(* Logix 5000 project; controller cal1615 1756-L62 rev 20.11; software revision 20.05; part 20 of 81 *)
(* tags used below, declared in another part *)
   AFI : BOOL;   // Always False Bit
   FAULT : BOOL;   // Fault AFI
   p01_param_open_oven_temp : REAL;
   p01_param_oven_timer_presets : DINT[32];   // System Parameter Oven Timer Presets
   p01_recipe_active : recipe;   // Active Recipe
   p01_sys_enc : SYS_ENC;   // System Encoder
   p01r09_open_oven : BOOL;
   p01r09_pb_global_reset : BOOL;   // System Modes PB: Global Fault Reset
   p01r13_permissive_oxidizer : BOOL;   // System Line Start Sequence Permissive Oxidizer
   p02_dint_from_hmi : hmi_dint;
   p11_ai_tc01 : REAL;   // Zone 1 Analog Input Control Thermocouple 1
   p11_ai_tc02 : REAL;   // Zone 1 Analog Input Control Thermocouple 2
   p11_di_burner_auto : BOOL;   // Zone 1 Digital Input Burner Auto
   p11_di_burner_safeties_ok : BOOL;   // Zone 1 Digital Input Burner Safeties Ok
   p11_di_exh_flow_ok : BOOL;   // Zone 1 Digital Input Exhaust Flow OK
   p11_di_flame_on : BOOL;   // Zone 1 Digital Input Burner is On
   p11_di_recirc_flow_ok : BOOL;   // Zone 1 Digital Input Recirc Flow OK
   p11_param_fast_to_soak : REAL;   // Zone 1 Parameter Fast to Soak Control
   p11_param_pid1_ff : REAL;   // Zone 1 Parameter Fast PID Bias
   p11_param_pid1_kd : REAL;   // Zone 1 Parameter Fast PID Derivative Gain
   p11_param_pid1_ki : REAL;   // Zone 1 Parameter Fast PID Integral Gain
   p11_param_pid1_kp : REAL;   // Zone 1 Parameter Fast PID Proportional Gain
   p11_param_soak_to_fast : REAL;   // Zone 1 Parameter Soak to Fast Control
   p11r01 : routine;   // Zone 1 Main
   p11r02_shutdown_temp : BOOL;   // Zone 1 Misc Control Safe Shutdown Temperature
   p11r02_timer_safe_temp : TIMER[2];   // Zone 1 Misc Control Chamber SafeTemperature Dwell
   p11r10 : routine;   // Zone 1
   p11r10_timer_fault : TIMER[4];   // Zone 1 Fault Delay
   p11r10_timer_warning : TIMER[4];   // Zone 1 Warning Delay
   p11r12_Oven_auto_run_on : BOOL;   // Zone 1 Temp Sequence Oven Auto Run On
   p11r20 : routine;   // Zone 1 Temp Sequence
   p11r20_safeties_ok : BOOL;   // Zone 1 Temperature Control Burner Safeties OK this Lightoff
   p11r20_state : DINT;   // Zone 1 Temperature Control State
   p11r20_status : DINT;   // Zone 1 Temperature Control Sequence Status
   p11r20_timer_fault : TIMER[4];   // Zone 1 Temp Sequence Fault Delay
   p11r20_timer_state_11 : TIMER;   // Zone 1 Temp Sequence State 11 Dwell
   p11r20_timer_state_3 : TIMER;   // Zone 1 Temperature Control State 3 Dwell
   p11r20_timer_state_4 : TIMER;   // Zone 1 Temp Sequence State 4 Dwell
   p11r20_timer_state_7 : TIMER;   // Zone 1 Temp Sequence State 7 Dwell
   p11r20_timer_warning : TIMER[4];   // Zone 1 Temp Sequence Warning Delay
   p11r30 : routine;   // Zone 1 Temperature Control
   p11r30_cv_man_sp : REAL;   // Zone 1 Temperature Control Manual Heat Control Valve Setpoint
   p11r30_pb_auto : BOOL;   // Zone 1 Temperature Control PB: Zone Control Auto
   p11r30_pb_manual : BOOL;   // Zone 1 Temperature Control PB: Zone Control Manual
   p11r30_pb_zone_off : BOOL;   // Zone 1 Temperature Control PB: Stop Zone Heat Control
   p11r30_pb_zone_on : BOOL;   // Zone 1 Temperature Control PB: Start Zone Heat Control
   p11r30_permissive_run : BOOL;   // Zone 1 Temperature Control Run Permissive
   p11r30_pid_temp : PID;   // Zone 1 Temperature Control PID
   p11r30_pid_temp_pv : REAL;   // Zone 1 Temperature Control PID Temp Process Variable
   p11r30_pid_temp_sp : REAL;   // Zone 1 Temperature Control PID Temperature Control Setpoint
   p11r30_pid_temp_sp_error : REAL;   // Zone 1 Temperature Control Setpoint/Process Variable Error (ABS)
   p11r30_pid_temp_sp_last : REAL;   // Zone 1 Temperature Control Setpoint Last Scan
   p11r30_request_deviation_warning : BOOL;   // Zone 1 Temperature Control Request Setpoint Deviation Warning
   p11r30_request_heat : BOOL;   // Zone 1 Temperature Control Request Heat
   p11r30_request_heat_last : BOOL;   // Zone 1 Temperature Control Request Heat Last Scan
   p11r30_request_manual : BOOL;   // Zone 1 Temperature Control Request Manual Control
   p11r30_request_PID_shot : BOOL;
   p11r30_request_soak_control : BOOL;   // Zone 1 Temperature Control Request Soak Control
   p11r30_temp_deviation_setpoint : DINT;
   p11r30_timer_warning : TIMER[12];   // Zone 1 Temperature Control Warning Delay
   p11r30_vfds_ok : BOOL;
   p11r31 : routine;   // Zone 1 Exhaust VFD
   p11r32 : routine;   // Zone 1 Recirc VFD
   p12r30 : routine;   // Zone 2 Temperature Control
   p23_di_impreg_exhaust_running : BOOL;
   p23_di_impreg_tank_up : BOOL;   // Input Impreg Dip Tank Up
   p23r02 : routine;   // Impreg Misc Control
   p23r13 : routine;
(* P11_Zone_1, continued *)

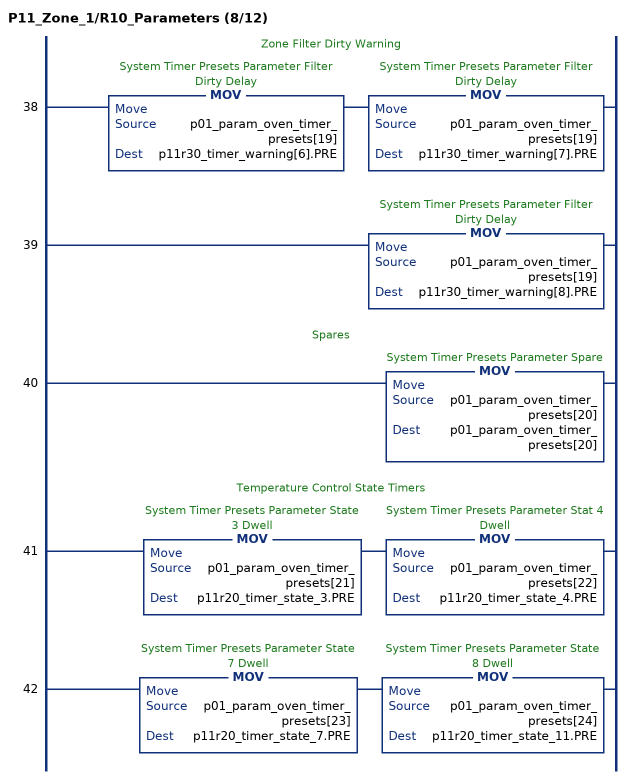
   [picture p305: P11_Zone_1/R10_Parameters rungs 38-42]
   // Zone Filter Dirty Warning
   38: MOV(p01_param_oven_timer_presets[19],p11r30_timer_warning[6].PRE)MOV(p01_param_oven_timer_presets[19],p11r30_timer_warning[7].PRE);
   39: MOV(p01_param_oven_timer_presets[19],p11r30_timer_warning[8].PRE);
   // Spares
   40: MOV(p01_param_oven_timer_presets[20],p01_param_oven_timer_presets[20]);
   // Temperature Control State Timers
   41: MOV(p01_param_oven_timer_presets[21],p11r20_timer_state_3.PRE)MOV(p01_param_oven_timer_presets[22],p11r20_timer_state_4.PRE);
   42: MOV(p01_param_oven_timer_presets[23],p11r20_timer_state_7.PRE)MOV(p01_param_oven_timer_presets[24],p11r20_timer_state_11.PRE);
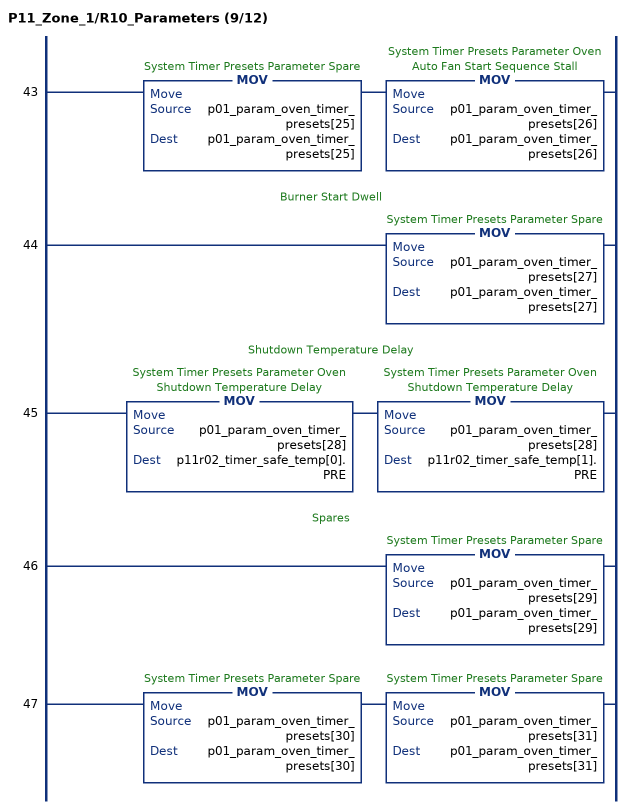
   43: MOV(p01_param_oven_timer_presets[25],p01_param_oven_timer_presets[25])MOV(p01_param_oven_timer_presets[26],p01_param_oven_timer_presets[26]);
   // Burner Start Dwell
   44: MOV(p01_param_oven_timer_presets[27],p01_param_oven_timer_presets[27]);
   // Shutdown Temperature Delay
   45: MOV(p01_param_oven_timer_presets[28],p11r02_timer_safe_temp[0].PRE)MOV(p01_param_oven_timer_presets[28],p11r02_timer_safe_temp[1].PRE);
   // Spares
   46: MOV(p01_param_oven_timer_presets[29],p01_param_oven_timer_presets[29]);
   47: MOV(p01_param_oven_timer_presets[30],p01_param_oven_timer_presets[30])MOV(p01_param_oven_timer_presets[31],p01_param_oven_timer_presets[31]);
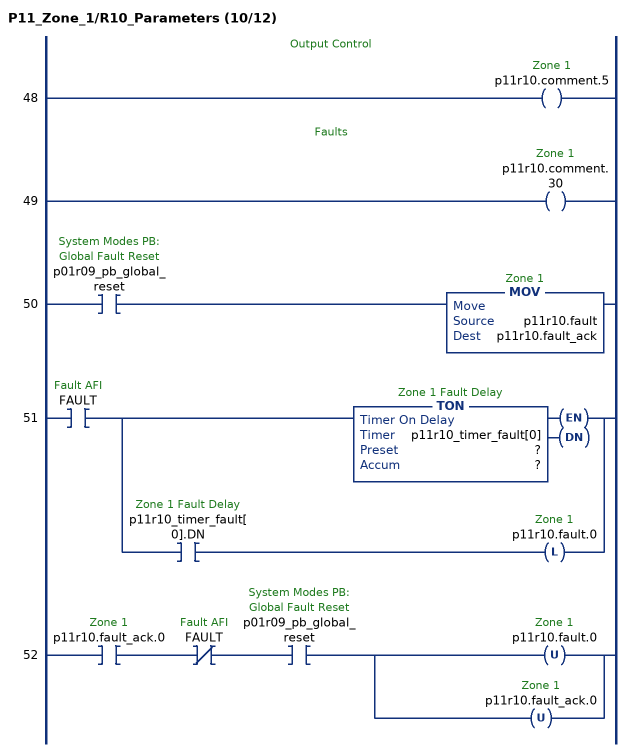
   // Output Control
   48: OTE(p11r10.comment.5);
   // Faults
   49: OTE(p11r10.comment.30);
   50: XIC(p01r09_pb_global_reset)MOV(p11r10.fault,p11r10.fault_ack);
   51: XIC(FAULT)[TON(p11r10_timer_fault[0],?,?) ,XIC(p11r10_timer_fault[0].DN) OTL(p11r10.fault.0) ];
   52: XIC(p11r10.fault_ack.0)XIO(FAULT)XIC(p01r09_pb_global_reset)[OTU(p11r10.fault.0) ,OTU(p11r10.fault_ack.0) ];
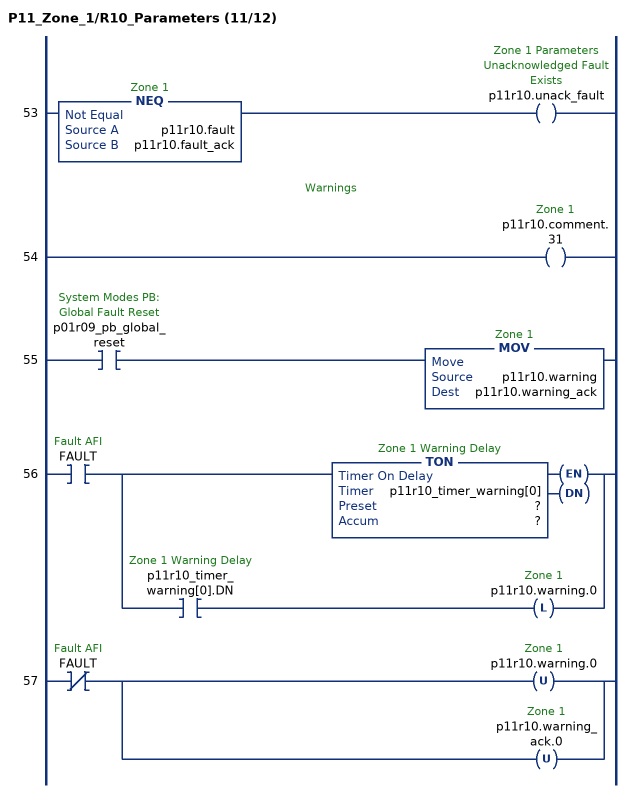
   53: NEQ(p11r10.fault,p11r10.fault_ack)OTE(p11r10.unack_fault);
   // Warnings
   54: OTE(p11r10.comment.31);
   55: XIC(p01r09_pb_global_reset)MOV(p11r10.warning,p11r10.warning_ack);
   56: XIC(FAULT)[TON(p11r10_timer_warning[0],?,?) ,XIC(p11r10_timer_warning[0].DN) OTL(p11r10.warning.0) ];
   57: XIO(FAULT)[OTU(p11r10.warning.0) ,OTU(p11r10.warning_ack.0) ];
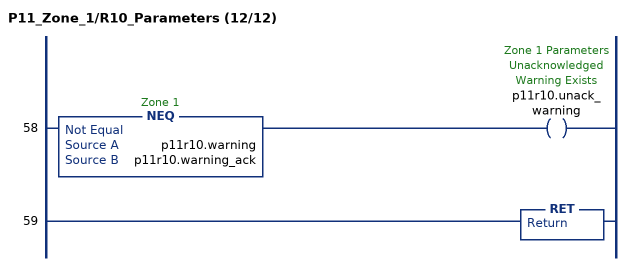
   58: NEQ(p11r10.warning,p11r10.warning_ack)OTE(p11r10.unack_warning);
   59: RET();
END_ROUTINE

ROUTINE R20_Temp_Sequence   (* ladder *)
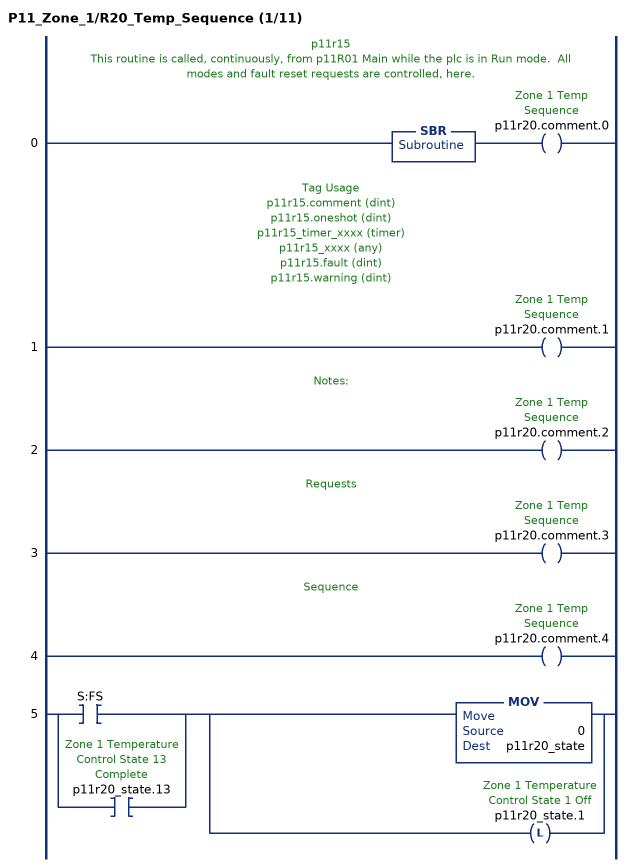
   // p11r15
   // This routine is called, continuously, from p11R01 Main while the plc is in Run mode.  All modes and fault reset requests are controlled, here.
   0: SBR()OTE(p11r20.comment.0);
   // Tag Usage
   // p11r15.comment (dint)
   // p11r15.oneshot (dint)
   // p11r15_timer_xxxx (timer)
   // p11r15_xxxx (any)
   // p11r15.fault (dint)
   // p11r15.warning (dint)
   1: OTE(p11r20.comment.1);
   // Notes:
   2: OTE(p11r20.comment.2);
   // Requests
   3: OTE(p11r20.comment.3);
   // Sequence
   4: OTE(p11r20.comment.4);
   5: [XIC(S:FS) ,XIC(p11r20_state.13) ][MOV(0,p11r20_state) ,OTL(p11r20_state.1) ];
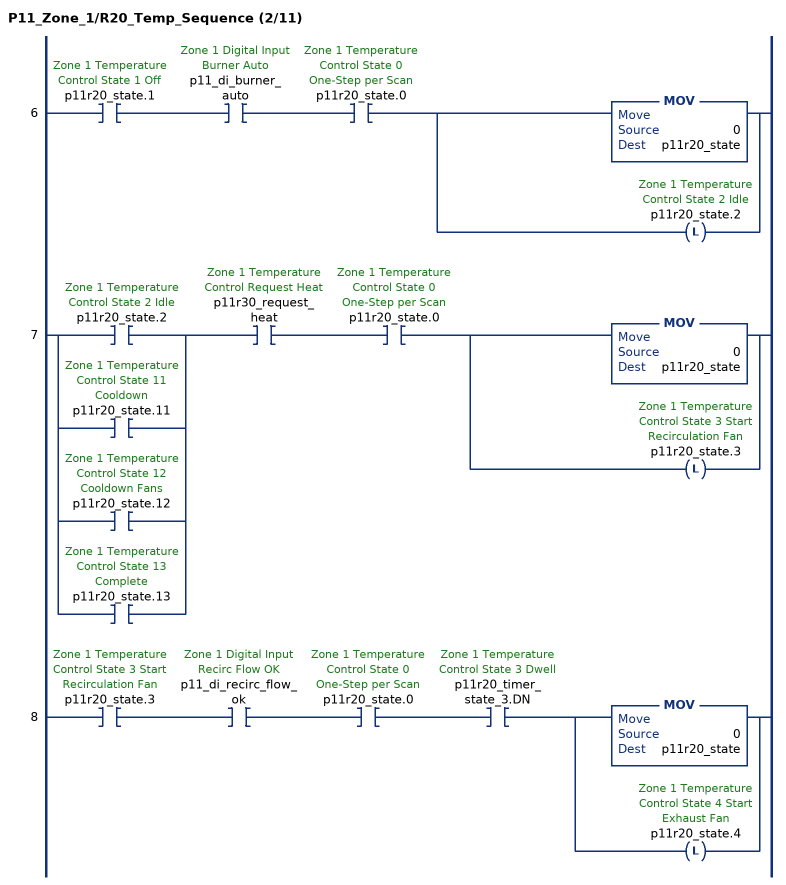
   6: XIC(p11r20_state.1)XIC(p11_di_burner_auto)XIC(p11r20_state.0)[MOV(0,p11r20_state) ,OTL(p11r20_state.2) ];
   7: [XIC(p11r20_state.2) ,XIC(p11r20_state.11) ,XIC(p11r20_state.12) ,XIC(p11r20_state.13) ]XIC(p11r30_request_heat)XIC(p11r20_state.0)[MOV(0,p11r20_state) ,OTL(p11r20_state.3) ];
   8: XIC(p11r20_state.3)XIC(p11_di_recirc_flow_ok)XIC(p11r20_state.0)XIC(p11r20_timer_state_3.DN)[MOV(0,p11r20_state) ,OTL(p11r20_state.4) ];
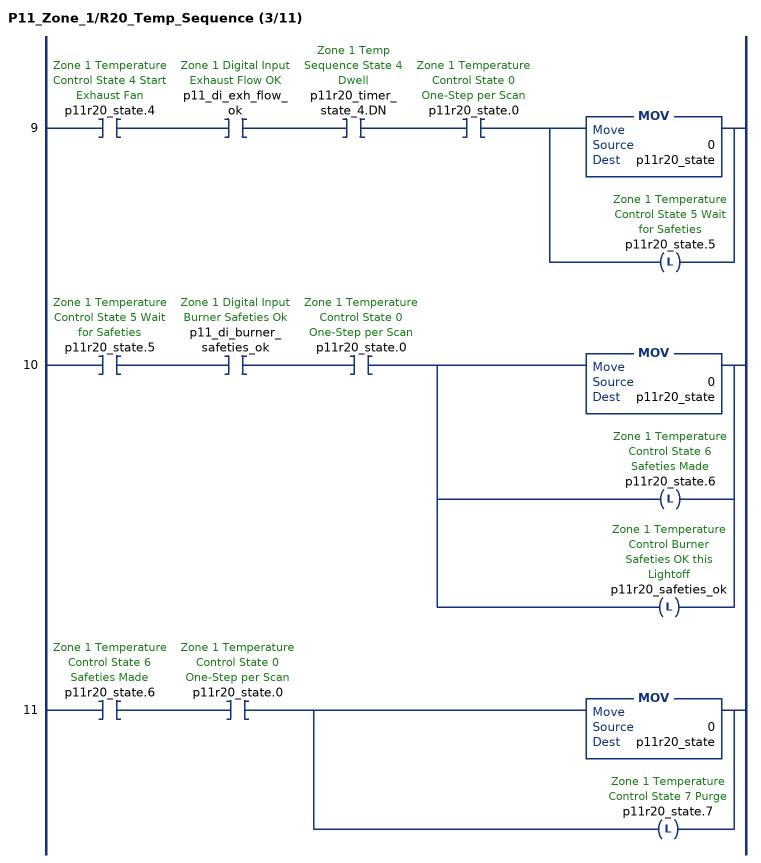
   9: XIC(p11r20_state.4)XIC(p11_di_exh_flow_ok)XIC(p11r20_timer_state_4.DN)XIC(p11r20_state.0)[MOV(0,p11r20_state) ,OTL(p11r20_state.5) ];
   10: XIC(p11r20_state.5)XIC(p11_di_burner_safeties_ok)XIC(p11r20_state.0)[MOV(0,p11r20_state) ,OTL(p11r20_state.6) ,OTL(p11r20_safeties_ok) ];
   11: XIC(p11r20_state.6)XIC(p11r20_state.0)[MOV(0,p11r20_state) ,OTL(p11r20_state.7) ];
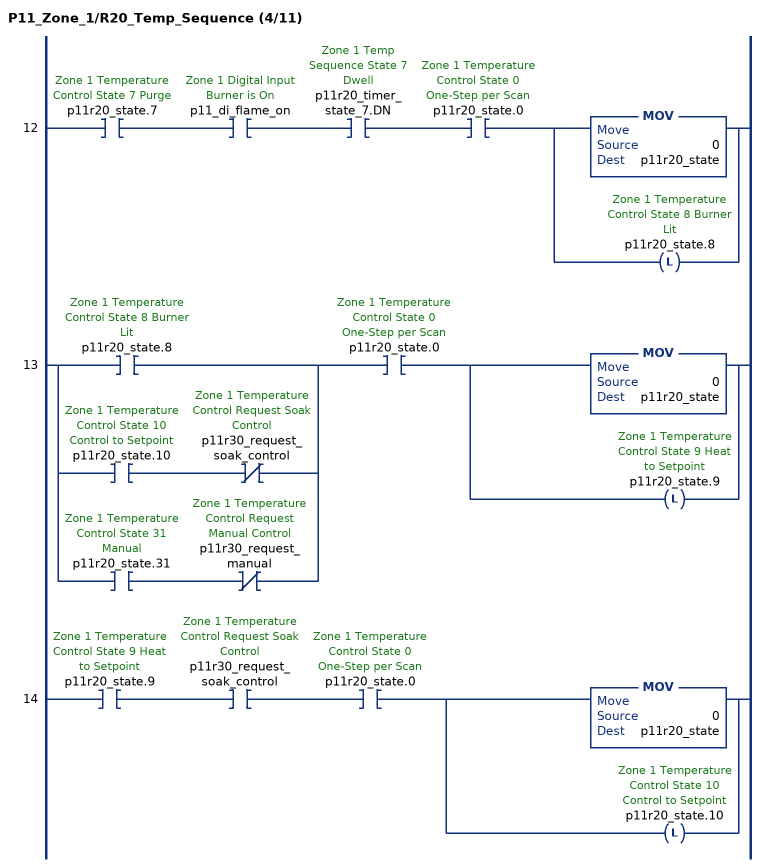
   12: XIC(p11r20_state.7)XIC(p11_di_flame_on)XIC(p11r20_timer_state_7.DN)XIC(p11r20_state.0)[MOV(0,p11r20_state) ,OTL(p11r20_state.8) ];
   13: [XIC(p11r20_state.8) ,XIC(p11r20_state.10) XIO(p11r30_request_soak_control) ,XIC(p11r20_state.31) XIO(p11r30_request_manual) ]XIC(p11r20_state.0)[MOV(0,p11r20_state) ,OTL(p11r20_state.9) ];
   14: XIC(p11r20_state.9)XIC(p11r30_request_soak_control)XIC(p11r20_state.0)[MOV(0,p11r20_state) ,OTL(p11r20_state.10) ];
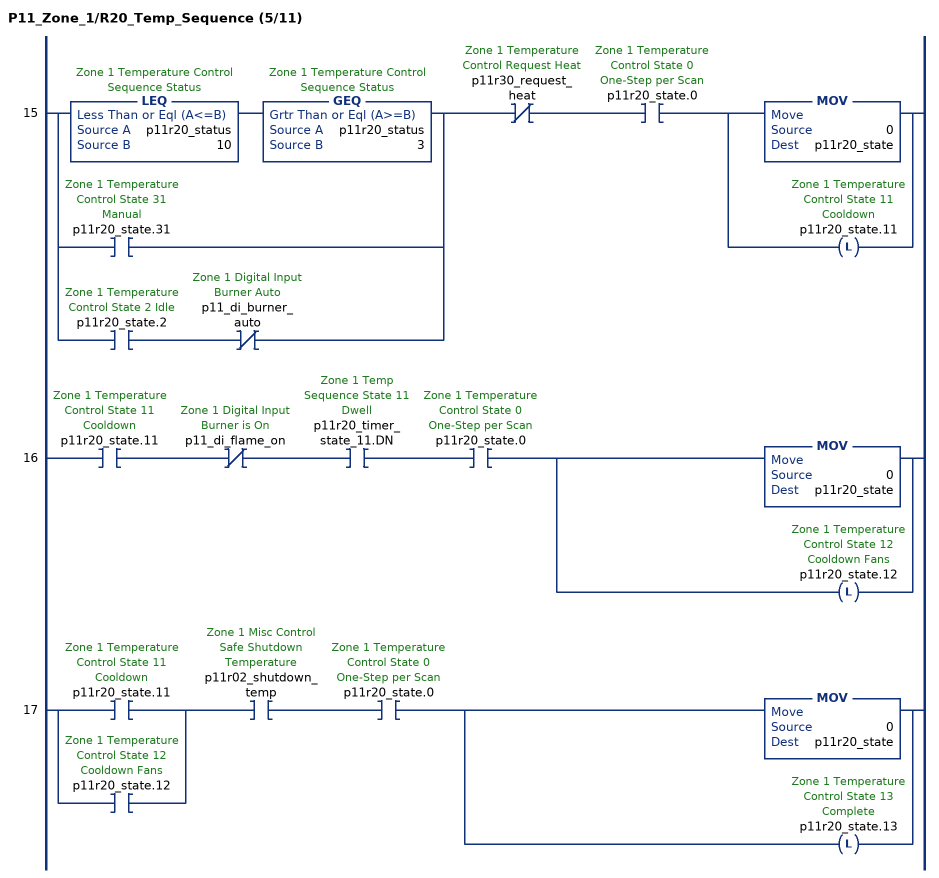
   15: [[LEQ(p11r20_status,10) GEQ(p11r20_status,3) ,XIC(p11r20_state.31) ] ,XIC(p11r20_state.2) XIO(p11_di_burner_auto) ]XIO(p11r30_request_heat)XIC(p11r20_state.0)[MOV(0,p11r20_state) ,OTL(p11r20_state.11) ];
   16: XIC(p11r20_state.11)XIO(p11_di_flame_on)XIC(p11r20_timer_state_11.DN)XIC(p11r20_state.0)[MOV(0,p11r20_state) ,OTL(p11r20_state.12) ];
   17: [XIC(p11r20_state.11) ,XIC(p11r20_state.12) ]XIC(p11r02_shutdown_temp)XIC(p11r20_state.0)[MOV(0,p11r20_state) ,OTL(p11r20_state.13) ];
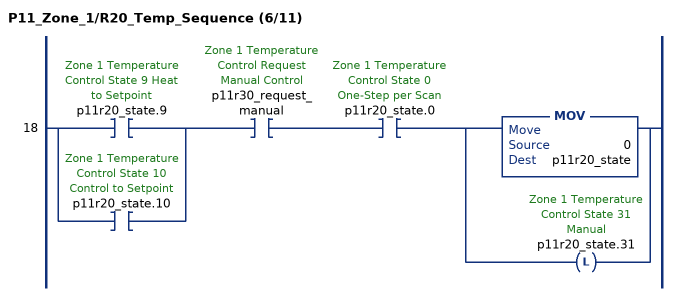
   18: [XIC(p11r20_state.9) ,XIC(p11r20_state.10) ]XIC(p11r30_request_manual)XIC(p11r20_state.0)[MOV(0,p11r20_state) ,OTL(p11r20_state.31) ];
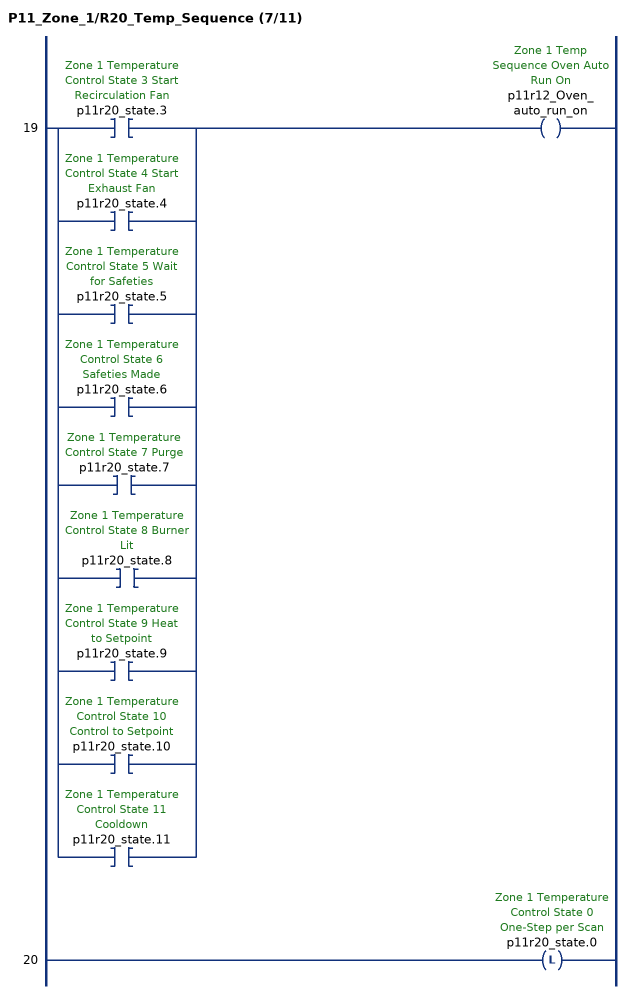
   19: [XIC(p11r20_state.3) ,XIC(p11r20_state.4) ,XIC(p11r20_state.5) ,XIC(p11r20_state.6) ,XIC(p11r20_state.7) ,XIC(p11r20_state.8) ,XIC(p11r20_state.9) ,XIC(p11r20_state.10) ,XIC(p11r20_state.11) ]OTE(p11r12_Oven_auto_run_on);
   20: OTL(p11r20_state.0);
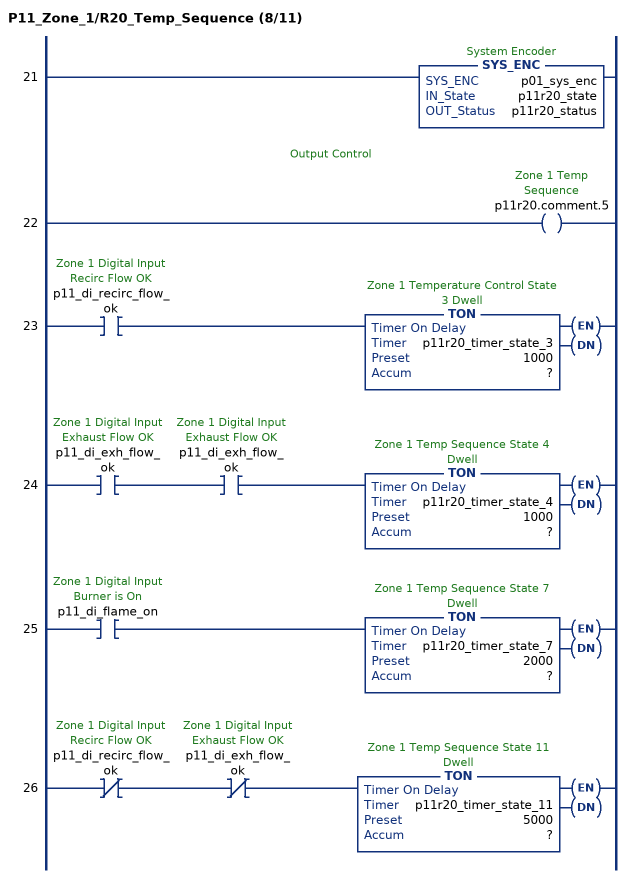
   21: SYS_ENC(p01_sys_enc,p11r20_state,p11r20_status);
   // Output Control
   22: OTE(p11r20.comment.5);
   23: XIC(p11_di_recirc_flow_ok)TON(p11r20_timer_state_3,?,?);
   24: XIC(p11_di_exh_flow_ok)XIC(p11_di_exh_flow_ok)TON(p11r20_timer_state_4,?,?);
   25: XIC(p11_di_flame_on)TON(p11r20_timer_state_7,?,?);
   26: XIO(p11_di_recirc_flow_ok)XIO(p11_di_exh_flow_ok)TON(p11r20_timer_state_11,?,?);
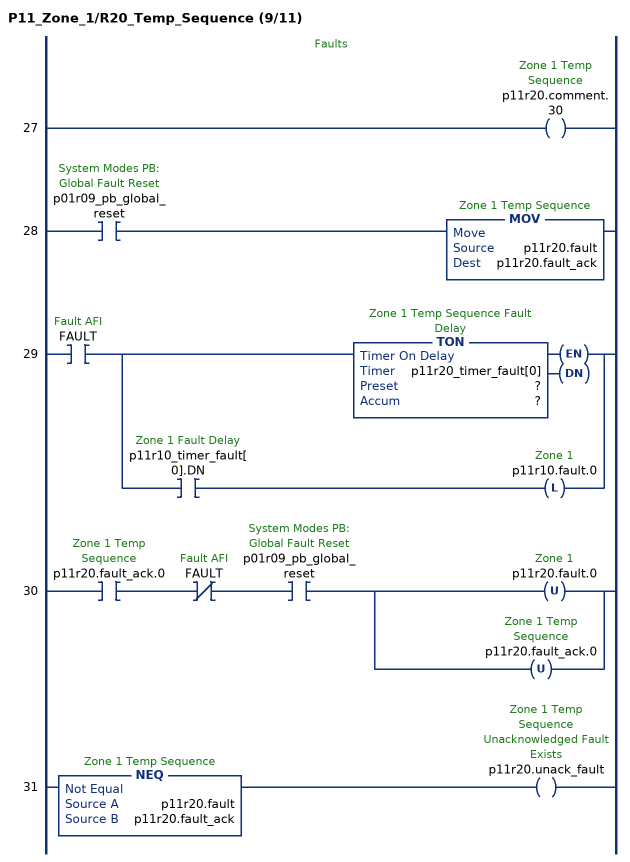
   // Faults
   27: OTE(p11r20.comment.30);
   28: XIC(p01r09_pb_global_reset)MOV(p11r20.fault,p11r20.fault_ack);
   29: XIC(FAULT)[TON(p11r20_timer_fault[0],?,?) ,XIC(p11r10_timer_fault[0].DN) OTL(p11r10.fault.0) ];
   30: XIC(p11r20.fault_ack.0)XIO(FAULT)XIC(p01r09_pb_global_reset)[OTU(p11r20.fault.0) ,OTU(p11r20.fault_ack.0) ];
   31: NEQ(p11r20.fault,p11r20.fault_ack)OTE(p11r20.unack_fault);
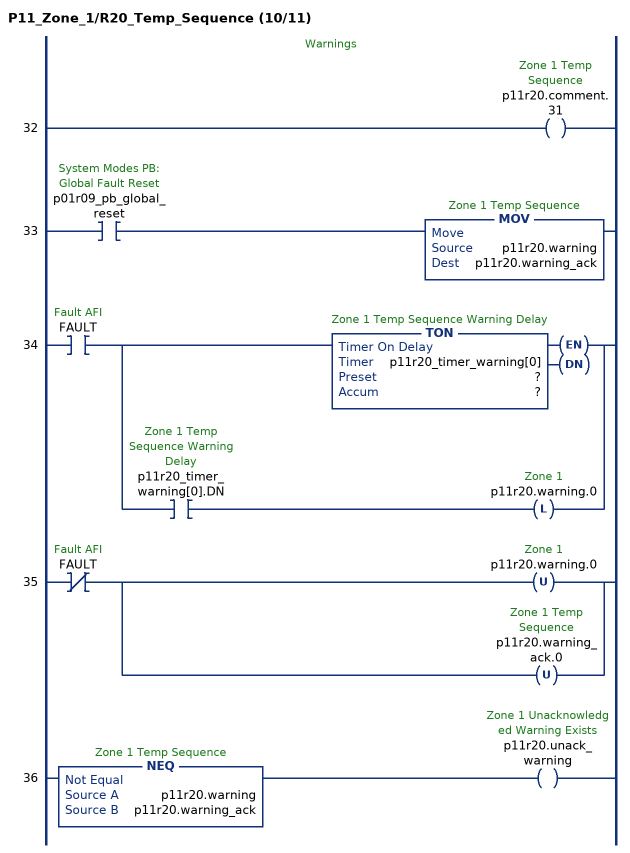
   // Warnings
   32: OTE(p11r20.comment.31);
   33: XIC(p01r09_pb_global_reset)MOV(p11r20.warning,p11r20.warning_ack);
   34: XIC(FAULT)[TON(p11r20_timer_warning[0],?,?) ,XIC(p11r20_timer_warning[0].DN) OTL(p11r20.warning.0) ];
   35: XIO(FAULT)[OTU(p11r20.warning.0) ,OTU(p11r20.warning_ack.0) ];
   36: NEQ(p11r20.warning,p11r20.warning_ack)OTE(p11r20.unack_warning);
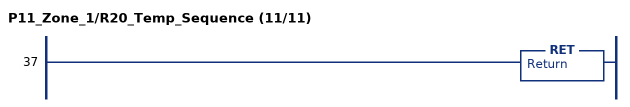
   37: RET();
END_ROUTINE

ROUTINE R30_Temperature_Control   (* ladder *)
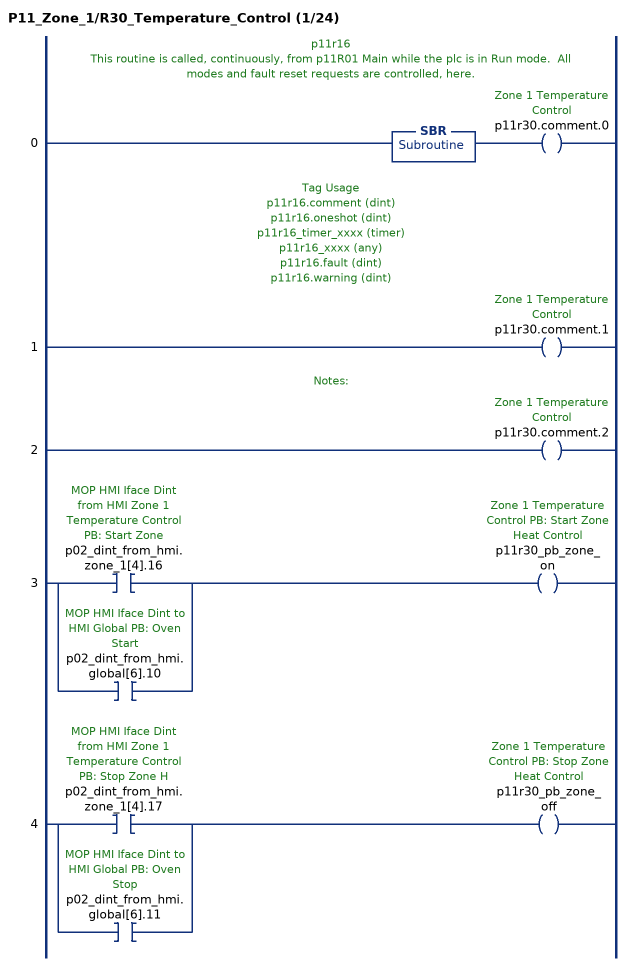
   // p11r16
   // This routine is called, continuously, from p11R01 Main while the plc is in Run mode.  All modes and fault reset requests are controlled, here.
   0: SBR()OTE(p11r30.comment.0);
   // Tag Usage
   // p11r16.comment (dint)
   // p11r16.oneshot (dint)
   // p11r16_timer_xxxx (timer)
   // p11r16_xxxx (any)
   // p11r16.fault (dint)
   // p11r16.warning (dint)
   1: OTE(p11r30.comment.1);
   // Notes:
   2: OTE(p11r30.comment.2);
   3: [XIC(p02_dint_from_hmi.zone_1[4].16) ,XIC(p02_dint_from_hmi.global[6].10) ]OTE(p11r30_pb_zone_on);
   4: [XIC(p02_dint_from_hmi.zone_1[4].17) ,XIC(p02_dint_from_hmi.global[6].11) ]OTE(p11r30_pb_zone_off);
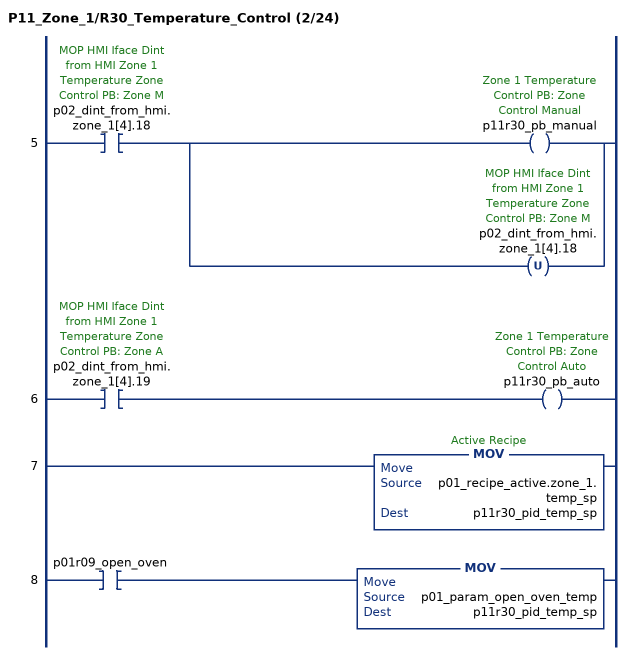
   5: XIC(p02_dint_from_hmi.zone_1[4].18)[OTE(p11r30_pb_manual) ,OTU(p02_dint_from_hmi.zone_1[4].18) ];
   6: XIC(p02_dint_from_hmi.zone_1[4].19)OTE(p11r30_pb_auto);
   7: MOV(p01_recipe_active.zone_1.temp_sp,p11r30_pid_temp_sp);
   8: XIC(p01r09_open_oven)MOV(p01_param_open_oven_temp,p11r30_pid_temp_sp);
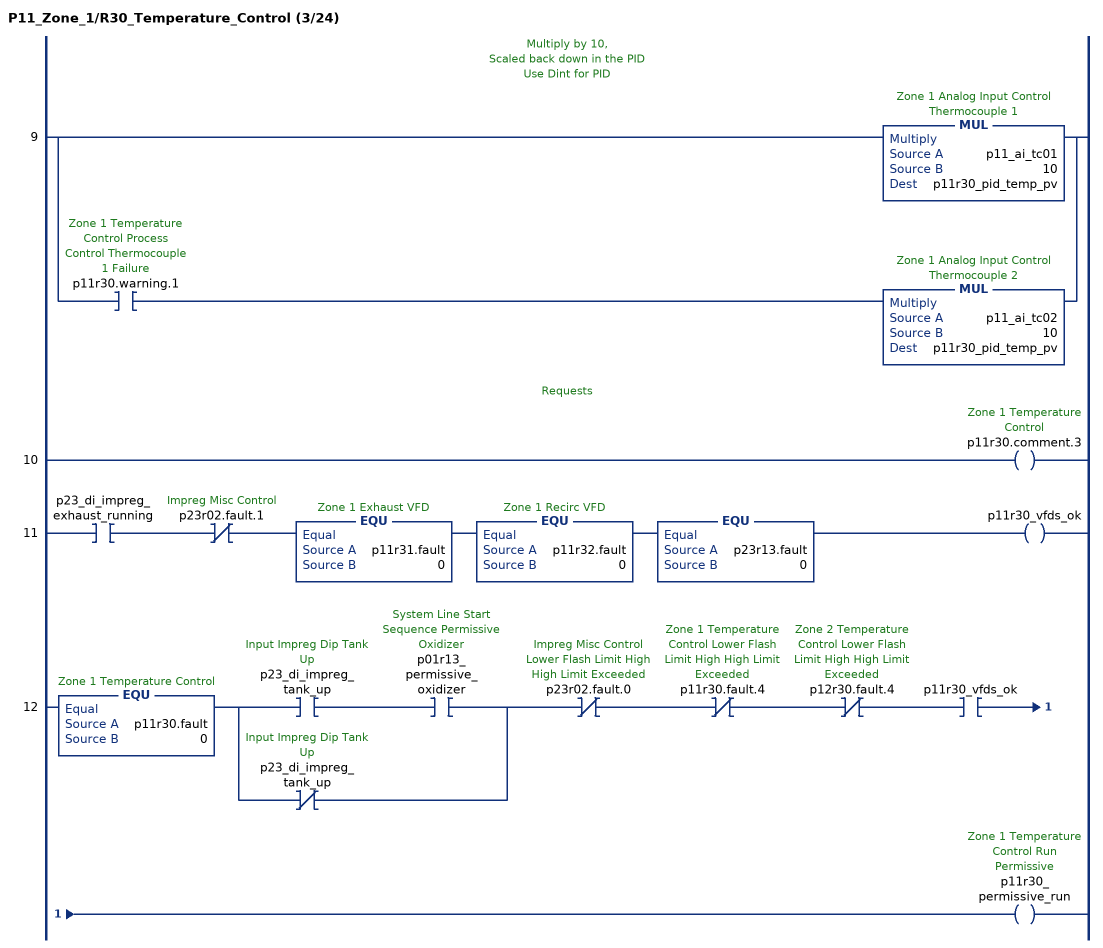
   // Multiply by 10,
   // Scaled back down in the PID
   // Use Dint for PID
   9: [MUL(p11_ai_tc01,10,p11r30_pid_temp_pv) ,XIC(p11r30.warning.1) MUL(p11_ai_tc02,10,p11r30_pid_temp_pv) ];
   // Requests
   10: OTE(p11r30.comment.3);
   11: XIC(p23_di_impreg_exhaust_running)XIO(p23r02.fault.1)EQU(p11r31.fault,0)EQU(p11r32.fault,0)EQU(p23r13.fault,0)OTE(p11r30_vfds_ok);
   12: EQU(p11r30.fault,0)[XIC(p23_di_impreg_tank_up) XIC(p01r13_permissive_oxidizer) ,XIO(p23_di_impreg_tank_up) ]XIO(p23r02.fault.0)XIO(p11r30.fault.4)XIO(p12r30.fault.4)XIC(p11r30_vfds_ok)OTE(p11r30_permissive_run);
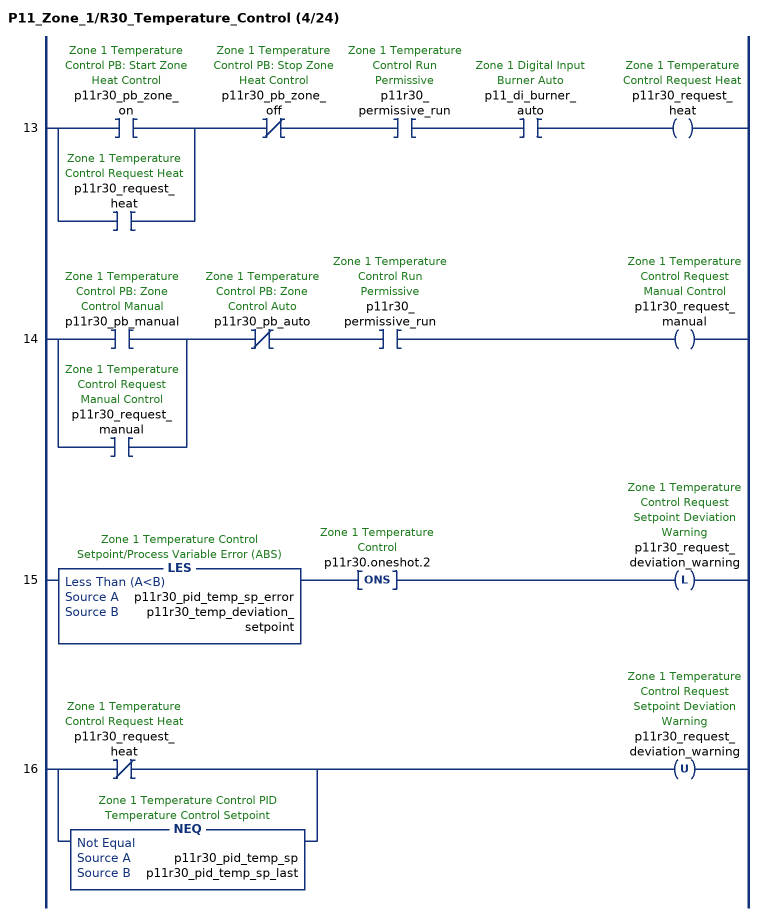
   13: [XIC(p11r30_pb_zone_on) ,XIC(p11r30_request_heat) ]XIO(p11r30_pb_zone_off)XIC(p11r30_permissive_run)XIC(p11_di_burner_auto)OTE(p11r30_request_heat);
   14: [XIC(p11r30_pb_manual) ,XIC(p11r30_request_manual) ]XIO(p11r30_pb_auto)XIC(p11r30_permissive_run)OTE(p11r30_request_manual);
   15: LES(p11r30_pid_temp_sp_error,p11r30_temp_deviation_setpoint)ONS(p11r30.oneshot.2)OTL(p11r30_request_deviation_warning);
   16: [XIO(p11r30_request_heat) ,NEQ(p11r30_pid_temp_sp,p11r30_pid_temp_sp_last) ]OTU(p11r30_request_deviation_warning);
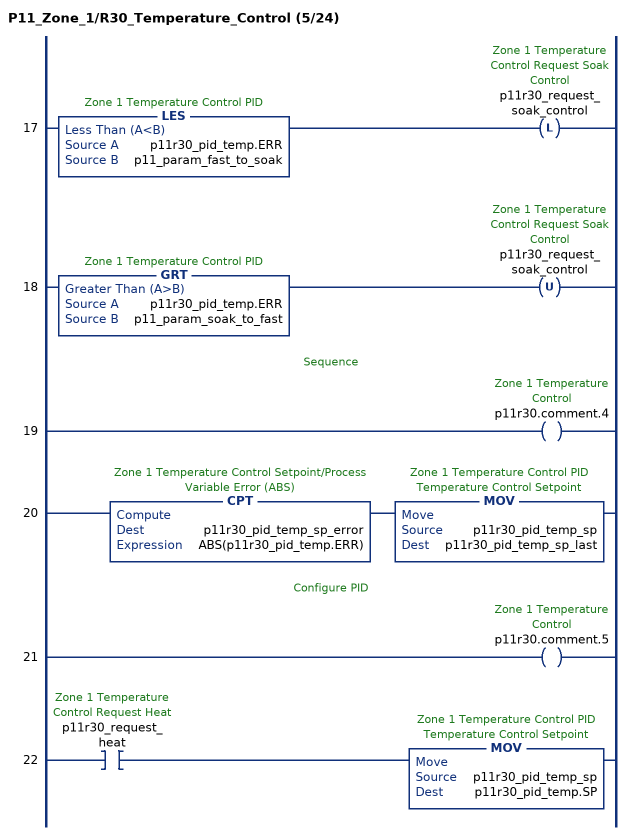
   17: LES(p11r30_pid_temp.ERR,p11_param_fast_to_soak)OTL(p11r30_request_soak_control);
   18: GRT(p11r30_pid_temp.ERR,p11_param_soak_to_fast)OTU(p11r30_request_soak_control);
   // Sequence
   19: OTE(p11r30.comment.4);
   20: CPT(p11r30_pid_temp_sp_error,ABS(p11r30_pid_temp.ERR))MOV(p11r30_pid_temp_sp,p11r30_pid_temp_sp_last);
   // Configure PID
   21: OTE(p11r30.comment.5);
   22: XIC(p11r30_request_heat)MOV(p11r30_pid_temp_sp,p11r30_pid_temp.SP);
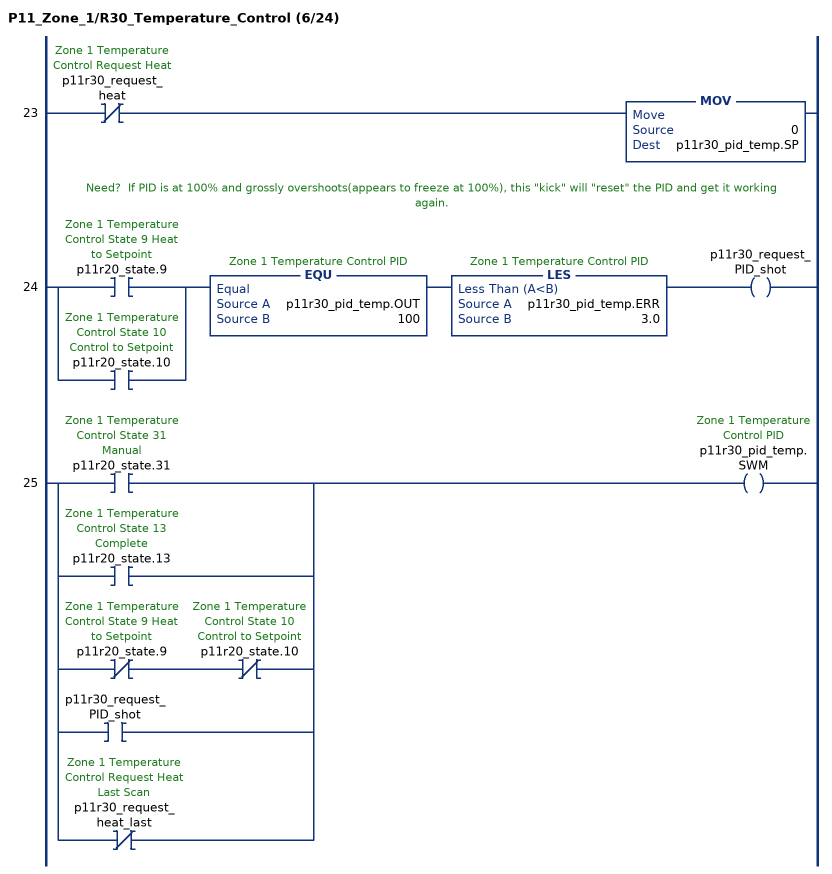
   23: XIO(p11r30_request_heat)MOV(0,p11r30_pid_temp.SP);
   // Need?  If PID is at 100% and grossly overshoots(appears to freeze at 100%), this "kick" will "reset" the PID and get it working again.
   24: [XIC(p11r20_state.9) ,XIC(p11r20_state.10) ]EQU(p11r30_pid_temp.OUT,100)LES(p11r30_pid_temp.ERR,3.0)OTE(p11r30_request_PID_shot);
   25: [XIC(p11r20_state.31) ,XIC(p11r20_state.13) ,XIO(p11r20_state.9) XIO(p11r20_state.10) ,XIC(p11r30_request_PID_shot) ,XIO(p11r30_request_heat_last) ]OTE(p11r30_pid_temp.SWM);
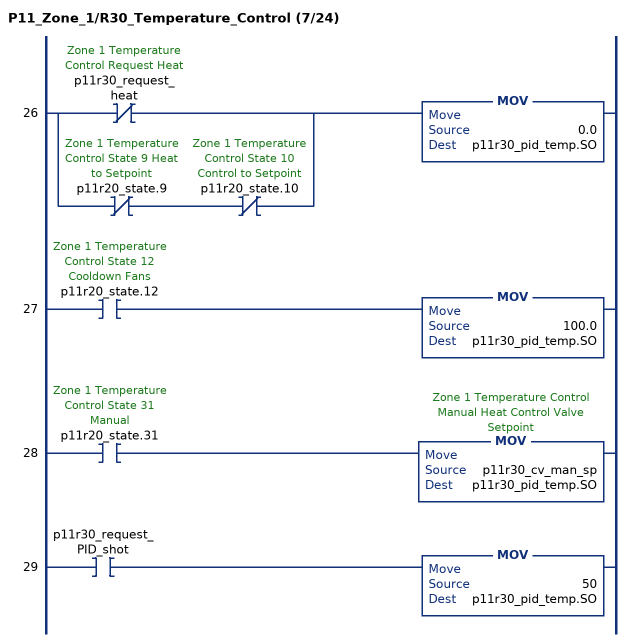
   26: [XIO(p11r30_request_heat) ,XIO(p11r20_state.9) XIO(p11r20_state.10) ]MOV(0.0,p11r30_pid_temp.SO);
   27: XIC(p11r20_state.12)MOV(100.0,p11r30_pid_temp.SO);
   28: XIC(p11r20_state.31)MOV(p11r30_cv_man_sp,p11r30_pid_temp.SO);
   29: XIC(p11r30_request_PID_shot)MOV(50,p11r30_pid_temp.SO);
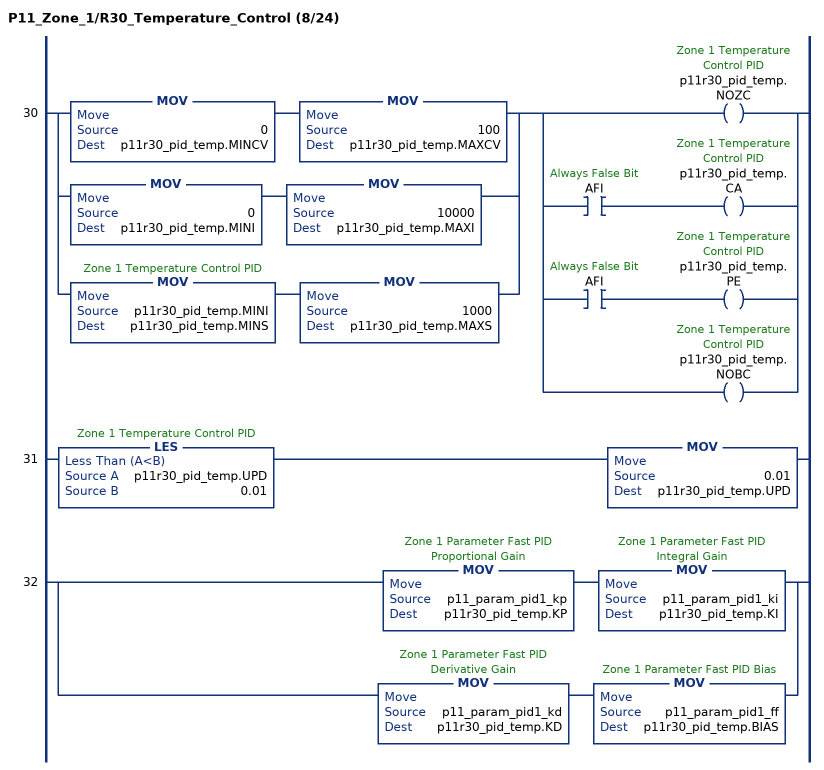
   30: [MOV(0,p11r30_pid_temp.MINCV) MOV(100,p11r30_pid_temp.MAXCV) ,MOV(0,p11r30_pid_temp.MINI) MOV(10000,p11r30_pid_temp.MAXI) ,MOV(p11r30_pid_temp.MINI,p11r30_pid_temp.MINS) MOV(1000,p11r30_pid_temp.MAXS) ][OTE(p11r30_pid_temp.NOZC) ,XIC(AFI) OTE(p11r30_pid_temp.CA) ,XIC(AFI) OTE(p11r30_pid_temp.PE) ,OTE(p11r30_pid_temp.NOBC) ];
   31: LES(p11r30_pid_temp.UPD,0.01)MOV(0.01,p11r30_pid_temp.UPD);
   32: [MOV(p11_param_pid1_kp,p11r30_pid_temp.KP) MOV(p11_param_pid1_ki,p11r30_pid_temp.KI) ,MOV(p11_param_pid1_kd,p11r30_pid_temp.KD) MOV(p11_param_pid1_ff,p11r30_pid_temp.BIAS) ];
